// TIA Portal V17 export
// export: Created 2024-08-26T21:10:48.3415038Z, ExportSetting WithDefaults, DisplayName Totally Integrated Automation Portal, DisplayVersion V17 Update 7, DisplayName TIA Portal Openness, DisplayVersion V17 Update 7, DisplayName TIA Portal Version Control Interface, DisplayVersion V17, DisplayName SINAMICS Startdrive Advanced, DisplayVersion V17 SP2, DisplayName SINAMICS Startdrive G110M, G120, G120C, G120D, G120P, G115D, DisplayVersion V17 SP2, DisplayName SINAMICS Startdrive G130, G150, S120, S150, SINAMICS MV, S210, DisplayVersion V17 SP2, DisplayName STEP 7 Professional, DisplayVersion V17 Update 7, DisplayName STEP 7 Safety, DisplayVersion V17 Update 6, DisplayName WinCC Advanced / Unified PC, DisplayVersion V17 Update 7
DATA_BLOCK "ALARM_DEVICE"   // DB37
{ S7_Optimized_Access := 'TRUE' }
VERSION : 0.1
// stored: AutoNumber true, DBAccessibleFromOPCUA true, DBAccessibleFromWebserver true, IsOnlyStoredInLoadMemory false, IsRetainMemResEnabled false, IsWriteProtectedInAS false, MemoryReserve 100
   VAR
      bannerStatus : Array[0..1023] of Bool;
      manifold : Array[0..1023] of Bool;
      iolink2 : Array[0..1023] of Bool;
      iolink1 : Array[0..1023] of Bool;
   END_VAR
BEGIN
   bannerStatus[0..1023] := FALSE;
   manifold[0..1023] := FALSE;
   iolink2[0] := TRUE;
   iolink2[1..5] := FALSE;
   iolink2[6] := TRUE;
   iolink2[7..1023] := FALSE;
   iolink1[0..1023] := FALSE;
END_DATA_BLOCK
